FUNCTION LPF_Function : REAL
VAR_INPUT
	SignalToFilter : REAL;
	FilterParams : POINTER TO LowPassFilter;
END_VAR
VAR
END_VAR

LPF_Function := FilterParams^.b0*SignalToFilter + FilterParams^.b1*FilterParams^.ErrorFilt - FilterParams^.OutputFilt*FilterParams^.a1;
FilterParams^.ErrorFilt := SignalToFilter;
FilterParams^.OutputFilt := LPF_Function;

END_FUNCTION

(* stored: Version 1.1.0.1, ProductVersion 3.1.4024.4
   POU LPF_Function: Id {999d823c-04f1-401e-8597-53114b0d73cd}, SpecialFunc None *)
